// TIA Portal V17 export
// export: Created 2022-04-06T07:28:40.36576Z, ExportSetting WithDefaults, DisplayName Totally Integrated Automation Portal, DisplayVersion V17, DisplayName TIA Portal Openness, DisplayVersion V17, DisplayName TIA Portal Version Control Interface, DisplayVersion V17, DisplayName TIA Portal Test Suite Advanced, DisplayVersion V17, DisplayName SINAMICS Startdrive Advanced, DisplayVersion V17, DisplayName SINAMICS Startdrive G130, G150, S120, S150, SINAMICS MV, S210, DisplayVersion V17, DisplayName SINAMICS Startdrive G110M, G120, G120C, G120D, G120P, G115D, DisplayVersion V17, DisplayName STEP 7 Professional, DisplayVersion V17, DisplayName STEP 7 Safety, DisplayVersion V17, DisplayName WinCC Advanced / Unified PC, DisplayVersion V17
VAR_GLOBAL   // PLC tag table "默认变量表"
   Tag_1 AT %M0.2 : Bool;
   System_Byte AT %MB1 : Byte;
   FirstScan AT %M1.0 : Bool;
   DiagStatusUpdate AT %M1.1 : Bool;
   AlwaysTRUE AT %M1.2 : Bool;
   AlwaysFALSE AT %M1.3 : Bool;
   Clock_Byte AT %MB0 : Byte;
   Clock_10Hz AT %M0.0 : Bool;
   Clock_5Hz AT %M0.1 : Bool;
   "Clock_2.5Hz" AT %M0.2 : Bool;
   Clock_2Hz AT %M0.3 : Bool;
   "Clock_1.25Hz" AT %M0.4 : Bool;
   Clock_1Hz AT %M0.5 : Bool;
   "Clock_0.625Hz" AT %M0.6 : Bool;
   "Clock_0.5Hz" AT %M0.7 : Bool;
   "PositioningAxis_1_Actor_Interface_AddressIn(8)" AT %I256.0 : "PD_TEL105_IN";
   "PositioningAxis_1_Actor_Interface_AddressOut(8)" AT %Q256.0 : "PD_TEL105_OUT";
   profiSafeCtrl1 AT %Q276.0 : "LDrvSafe_typeSinaTlg901Control";
   proSafeStatus1 AT %I276.0 : "LDrvSafe_typeSinaTlg901Status";
   profiSafeCtrl2 AT %Q310.0 : "LDrvSafe_typeSinaSTlg30Control";
   profiSafeStatus2 AT %I310.0 : "LDrvSafe_typeSinaSTlg30Status";
   "PositioningAxis_2_Actor_Interface_AddressIn(7)" AT %I290.0 : "PD_TEL105_IN";
   "PositioningAxis_2_Actor_Interface_AddressOut(7)" AT %Q290.0 : "PD_TEL105_OUT";
END_VAR
